FUNCTION_BLOCK FB_04
VAR_INPUT
END_VAR
VAR_OUTPUT
END_VAR
VAR
END_VAR

END_FUNCTION_BLOCK

(* stored: Version 1.1.0.1, ProductVersion 3.1.4024.12
   POU FB_04: Id {61a45d04-de20-40a0-a3b4-baa39636d5f6}, SpecialFunc None *)
